// SIMATIC STEP 7 (V5.x) project fh_config
// station: Hardware
// station: SIMATIC 300(1)
// station: P_ADR_BUS
// station: P_ADR_BUS
// station: Konfiguration
// program: S7-Programm

SYMBOL_TABLE
"Quader"	FC 1	FC 1
END_SYMBOL_TABLE

FUNCTION "Quader" : INT	// FC 1
VERSION : 0.1
VAR_INPUT
  Laenge : INT ;
  Breite : INT ;
  Hoehe : INT ;
END_VAR
VAR_OUTPUT
  RET_VAL : INT ;
END_VAR
VAR_TEMP
  Flaeche : INT ;
END_VAR
BEGIN
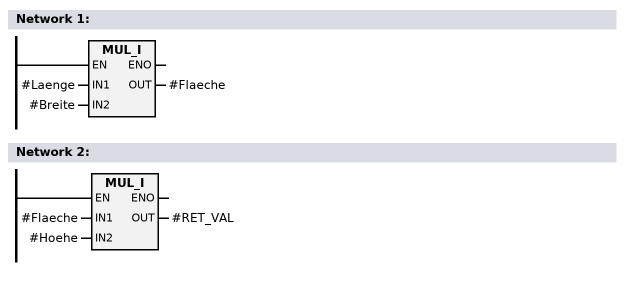
NETWORK
TITLE =
      L     #Laenge;
      L     #Breite;
      *I;
      T     #Flaeche;
      NOP   0;
NETWORK
TITLE =
      L     #Flaeche;
      L     #Hoehe;
      *I;
      T     #RET_VAL;
      NOP   0;
END_FUNCTION

ORGANIZATION_BLOCK OB 1
TITLE = "Main Program Sweep (Cycle)"
VERSION : 0.1
VAR_TEMP
  OB1_EV_CLASS : BYTE ;	//Bits 0-3 = 1 (Coming event), Bits 4-7 = 1 (Event class 1)
  OB1_SCAN_1 : BYTE ;	//1 (Cold restart scan 1 of OB 1), 3 (Scan 2-n of OB 1)
  OB1_PRIORITY : BYTE ;	//Priority of OB Execution
  OB1_OB_NUMBR : BYTE ;	//1 (Organization block 1, OB1)
  OB1_RESERVED_1 : BYTE ;	//Reserved for system
  OB1_RESERVED_2 : BYTE ;	//Reserved for system
  OB1_PREV_CYCLE : INT ;	//Cycle time of previous OB1 scan (milliseconds)
  OB1_MIN_CYCLE : INT ;	//Minimum cycle time of OB1 (milliseconds)
  OB1_MAX_CYCLE : INT ;	//Maximum cycle time of OB1 (milliseconds)
  OB1_DATE_TIME : DATE_AND_TIME ;	//Date and time OB1 started
END_VAR
BEGIN
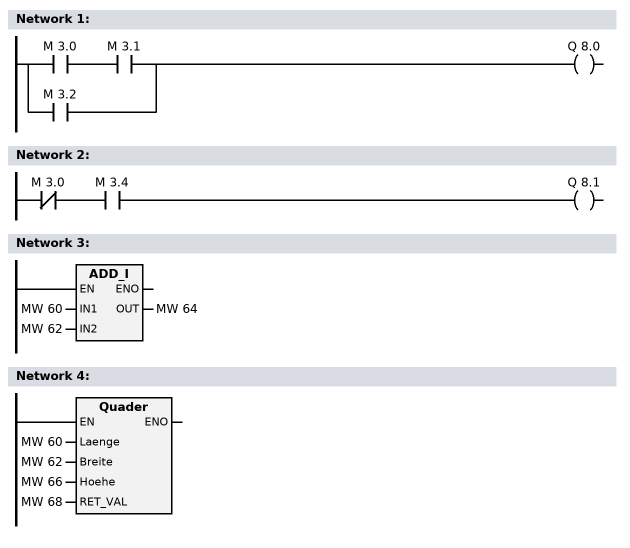
NETWORK
TITLE =
      A     M 3.0;
      A     M 3.1;
      O     M 3.2;
      =     Q 8.0;
NETWORK
TITLE =
      AN    M 3.0;
      A     M 3.4;
      =     Q 8.1;
NETWORK
TITLE =
      L     MW 60;
      L     MW 62;
      +I;
      T     MW 64;
      NOP   0;
NETWORK
TITLE =
      CALL  "Quader" (
           Laenge                   := MW 60,
           Breite                   := MW 62,
           Hoehe                    := MW 66,
           RET_VAL                  := MW 68);
      NOP   0;
END_ORGANIZATION_BLOCK
